Fanuc KAREL source: kt00407.KL

-- PROVISIONAL review KL for V770-1; original PC SHA256 62a5fcd888ec22cb1ca1c282bca46d6adcd652bda3282e239d83bd73776a724f
-- Incomplete behavior may be omitted. Consult companion uncertainty JSON. Do not deploy.
PROGRAM KT00407
%NOLOCKGROUP
VAR
  R1 : REAL
  OUT : BOOLEAN
-- UNRESOLVED_DECL Y2 type=002018
BEGIN
  -- UNRESOLVED_PC offsets 5-16; opcodes 2E,23
  -- UNRESOLVED_PC offsets 21-35; opcodes 2E,22,9D,33,B2
  -- UNRESOLVED_PC offsets 40-63; opcodes 21,22,9D,33,B1,64,71,23
  -- UNRESOLVED_PC offsets 68-72; opcodes 7F
END KT00407
